/// This function block is a container for all linked units that are used by this unit.
/// Linked units can be addressed through their individual interface.
FUNCTION_BLOCK TransportLinkedUnit EXTENDS TransportContainer
VAR_INPUT
  Assembly : IAssembly := ZModuleProgram.Assembly;
  Drilling : IDrilling := ZModuleProgram.Drilling;
  QualityInspection : IQualityInspection := ZModuleProgram.QualityInspection;
{attribute '__ZwPlcUnitEquipmentDeclaration__'} // Do not remove this attribute! It is used for code generation.
END_VAR

IF _isInitialized
THEN
  RETURN;
END_IF

{attribute '__ZwPlcUnitEquipmentImplementation__'} // Do not remove this attribute! It is used for code generation.

_isInitialized := TRUE;

END_FUNCTION_BLOCK

(* stored: Version 1.1.0.1
   POU TransportLinkedUnit: Id {72dc7f67-ee36-44b1-8aec-106abc2342c7}, SpecialFunc None *)
